// TIA Portal project "1212_test_signal_loadcell" (V17)

(* hardware
DEVICE "S7-1200 station_1"  S7-1200 Station
   slot 0: "Rack_0"  S7-1200 Rack  Rack  V1.0
   slot 1: "PLC_1"  CPU 1212C DC/DC/DC  6ES7 212-1AE40-0XB0  V4.2
DEVICE "PC-System_1"  SIMATIC PC station
   slot 0: "SIMATIC PC station"  Rail  SIMATIC PC-Station  V1.0
      slot 125: "Stationmanager"  Station_Manager  V6.0.4
   slot 1: "HMI_RT_1"  WinCC RT Advanced  6AV2 104-0xxxx-xxxx  17.0.0.0
      slot 33792: "Computer interface"  Host interface
*)

// ===== PLC "PLC_1"  CPU 1212C DC/DC/DC =====

VAR_GLOBAL   // PLC tag table "Default tag table"
   "sensor_input" AT %IW64 : Int;
   "Tag_2" AT %MD20 : Real;
   "KL_VAT" AT %MD30 : Real;
   "Tag_3" AT %MD110 : Real;
   "Tag_4" AT %MD120 : Real;
   "Tag_5" AT %MD130 : Real;
END_VAR

ORGANIZATION_BLOCK "Main"   // OB1, LAD, ProgramCycle
TITLE = "Main Program Sweep (Cycle)"
{ S7_Optimized_Access := 'TRUE' }
VERSION : 0.1
   VAR_INPUT
      Initial_Call : Bool;   // Initial call of this OB
      Remanence : Bool;   // =True, if remanent data are available
   END_VAR
BEGIN

REGION Network 1
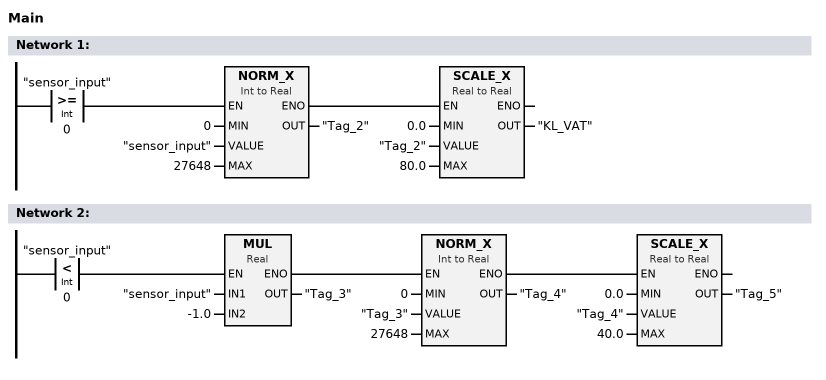
   RUNG wire#powerrail
      { S7_Templates := "SrcType := Int" } GE_Contact(in1 := "sensor_input", in2 := 0)
      { S7_Templates := "[SrcType := Int, DestType := Real]" } Normalize(min := 0, value := "sensor_input", max := 27648, out => "Tag_2")
      { S7_Templates := "[SrcType := Real, DestType := Real]" } Scale(min := 0.0, value := "Tag_2", max := 80.0, out => "KL_VAT")
   END_RUNG
   // the same network as SCL:
   IF "sensor_input" >= 0 THEN
       "Tag_2" := NORM_X(MIN := 0, VALUE := "sensor_input", MAX := 27648);
       "KL_VAT" := SCALE_X(MIN := 0.0, VALUE := "Tag_2", MAX := 80.0);
   END_IF;
END_REGION

REGION Network 2
   RUNG wire#powerrail
      { S7_Templates := "SrcType := Int" } LT_Contact(in1 := "sensor_input", in2 := 0)
      { S7_Templates := "SrcType := Real" } Mul(in1 := "sensor_input", in2 := -1.0, out => "Tag_3")
      { S7_Templates := "[SrcType := Int, DestType := Real]" } Normalize(min := 0, value := "Tag_3", max := 27648, out => "Tag_4")
      { S7_Templates := "[SrcType := Real, DestType := Real]" } Scale(min := 0.0, value := "Tag_4", max := 40.0, out => "Tag_5")
   END_RUNG
   // the same network as SCL:
   IF "sensor_input" < 0 THEN
       "Tag_3" := "sensor_input" * (-1.0);
       "Tag_4" := NORM_X(MIN := 0, VALUE := "Tag_3", MAX := 27648);
       "Tag_5" := SCALE_X(MIN := 0.0, VALUE := "Tag_4", MAX := 40.0);
   END_IF;
END_REGION
END_ORGANIZATION_BLOCK